FUNCTION_BLOCK Temperature_Transducer
VAR_INPUT
	RawValue			:	INT			:=	0;
	InstrumentEnable	:	BOOL		:=	TRUE;
END_VAR
VAR_OUTPUT
	Temperature_SI		:	REAL		:=	0.0;			//	°C
END_VAR
VAR
	Low_Alarm			:	BOOL		:=	FALSE;
	High_Alarm			:	BOOL		:=	FALSE;
	
	Low_Alarm_Setpoint	:	REAL		:=	0.000;			//	°C
	High_Alarm_Setpoint	:	REAL		:=	100.0;			//	°C
END_VAR

IF(InstrumentEnable)THEN
	Temperature_SI		:=	INT_TO_REAL(RawValue)/ 100.0;	//	Assumes That An EL3202 16-Bit RTD IO Card Is Used To Read The PT100 Instrument

	//	Alarm Functionality: Rising Edge Required For Event System To Trigger An Alarm Event
	IF(Temperature_SI < Low_Alarm_Setpoint)THEN
		Low_Alarm		:=	TRUE;
	ELSE
		Low_Alarm		:=	FALSE;
	END_IF;

	IF(Temperature_SI > High_Alarm_Setpoint)THEN
		Low_Alarm		:=	TRUE;
	ELSE
		Low_Alarm		:=	FALSE;
	END_IF;
ELSE
	Temperature_SI		:=	0.0;
END_IF;

END_FUNCTION_BLOCK

(* stored: Version 1.1.0.1, ProductVersion 3.1.4024.15
   POU Temperature_Transducer: Id {a55371ea-bc2e-480d-8efe-92c265429ebd}, SpecialFunc None *)
